Staubli VAL3: math.dtx

num nResult
num nIndex
num nResult2
num nTest[7]
num nResultTest
